(* CODESYS project sps_modbus_test_marcel_home.ecp

Project tree, tasks and I/O mapping:
  PFC200_2ETH_CAN_T : 750-8203 PFC200 2ETH CAN, WAGO, order no. 0750-8203, version 5.11.1.16
    application EM2MODBUSTESTMARCELHOME
      libraries: ; WagoAppPlcModbus, * (WAGO)
      task PLC_Task (cyclic, interval t#50ms, priority 15) calls PLC_PRG
      program PLC_PRG [ST]
    DeviceAdapter
    Kbus : Kbus, WAGO, version 1.4.0.2
        unmapped channels: K-BUS diagnostics
    MODBUS
      MODBUS : MODBUS, WAGO, order no. n/a, version 1.1.1.15
    CANbus
*)

// PFC200_2ETH_CAN_T/EM2MODBUSTESTMARCELHOME/PLC_PRG
PROGRAM PLC_PRG
VAR
	modbusServer: FbMbSimpleServertcp :=( xOpen := TRUE,
				wPort := 5020,
				utKeepAlive := (xEnable := TRUE,
						tMaxIdleTime := T#5S,
						tInterval := T#2S,
						udiProbes := 5
						),
				bUnitId := 1
				);
	myCoils : ARRAY[0..20] OF BOOL;
	myDiscreteInputs : ARRAY[0..148] OF BOOL;
	myInputRegisters : ARRAY[0..48] OF WORD;
	myHoldingRegisters : ARRAY[0..52] OF WORD;
	connected: BOOL := FALSE;
END_VAR

// Taster Control Unit auslesen.
// =============================
modbusServer( axDiscreteInputs := myDiscreteInputs,
			axCoils := myCoils,
			awInputRegisters := myInputRegisters,
			awHoldingRegisters := myHoldingRegisters
);
connected := modbusServer.udiConnectedClients > 0;
IF connected THEN
	//GVL_BRAKE.LEVEL :=  WORD_TO_INT(myHoldingRegisters[0]) - 1000;
	//GVL_TRACTION.IN_STROM := WORD_TO_INT(myHoldingRegisters[1]);//-1000
	//GVL_TRACTION.FAHRTRICHTUNG := myCoils[1];
	//GVL.HUPE := myCoils[6];
	//GVL_BRAKE.KOMPRESSOR := myCoils[8];
	
	//myInputRegisters[1] := REAL_TO_WORD(GVL_ENERGY.BAT0_CURRENT * 100);
	//myInputRegisters[2] := EMERGENCY_CONTROL.ErrorCode;
	//myInputRegisters[3] := REAL_TO_WORD(GVL_TRACTION.V_MEAN * 100);
	//myInputRegisters[4] := REAL_TO_WORD(GVL_BRAKE.KOMPRESSORDRUCK * 100);
	//myInputRegisters[5] := REAL_TO_WORD(GVL_BRAKE.BREMSDRUCK_1 * 100);
	//myInputRegisters[6] := REAL_TO_WORD(GVL_BRAKE.BREMSDRUCK_2 * 100);
	
	myDiscreteInputs[21] := FALSE;
	myDiscreteInputs[22] := FALSE;
	myDiscreteInputs[23] := FALSE;
	myDiscreteInputs[24] := FALSE;
	myDiscreteInputs[25] := myCoils[8];
	myDiscreteInputs[26] := myCoils[6];
	myDiscreteInputs[27] := TRUE;
	
	myInputRegisters[21] := 223;
	myInputRegisters[22] := 224;
	myInputRegisters[23] := 206;
	myInputRegisters[24] := 0;
	myInputRegisters[25] := 0;
	myInputRegisters[26] := 227;
	myInputRegisters[27] := 0;
	myInputRegisters[28] := 263;
	myInputRegisters[29] := 1869;
	myInputRegisters[30] := 0;
	myInputRegisters[31] := 0;
	myInputRegisters[32] := 235;
	myInputRegisters[33] := 120;
	myInputRegisters[34] := 5;
	myInputRegisters[35] := 0;
	myInputRegisters[36] := 239;
	myInputRegisters[37] := 0;
	myInputRegisters[38] := 0;
	myInputRegisters[39] := 238;
	myInputRegisters[40] := 211;
	myInputRegisters[41] := 1;
	myInputRegisters[42] := 36;
	myInputRegisters[43] := 225;
	myInputRegisters[44] := 0;
	myInputRegisters[45] := 0;
	myInputRegisters[46] := 226;
	
	
	
	
END_IF

END_PROGRAM
